// TwinCAT 3 PLC project PLC
// ProgramVersion: 3.1.4023.0
// libraries:
//   Lynus Communicator V2, * (Lynus AG)
//   Lynus Energy Basic, * (Lynus AG)
//   Lynus Energy ModbusTCP, * (Lynus AG)
//   Lynus Persistent Data V1, * (Lynus AG)
//   Tc2_Standard, * (Beckhoff Automation GmbH)
//   Tc2_System, * (Beckhoff Automation GmbH)
//   Tc3_Module, * (Beckhoff Automation GmbH)
// project tree:
//   / Fast.TcTTO, PlcTask.TcTTO, Slow.TcTTO
//   POUs/ prgCom.TcPOU, prgCS1.TcPOU, prgEMS.TcPOU, prgGrid.TcPOU, prgPD.TcPOU, prgVar.TcPOU
// real-time tasks:
//   TASK PlcTask: cycle T#10ms, priority 8, ADS port 350
//   TASK Fast: cycle T#5ms, priority 6, ADS port 351
//   TASK Slow: cycle T#20ms, priority 10, ADS port 352

CONFIGURATION PLC
    RESOURCE PLC ON TwinCAT3
        TASK Fast(INTERVAL := T#5ms, PRIORITY := 6);
        TASK PlcTask(INTERVAL := T#10ms, PRIORITY := 8);
        TASK Slow(INTERVAL := T#20ms, PRIORITY := 10);
        PROGRAM prgVar WITH Fast : prgVar;
        PROGRAM prgPD WITH PlcTask : prgPD;
        PROGRAM prgGrid WITH PlcTask : prgGrid;
        PROGRAM prgEMS WITH PlcTask : prgEMS;
        PROGRAM prgCS1 WITH PlcTask : prgCS1;
        PROGRAM prgCom WITH Slow : prgCom;
    END_RESOURCE
END_CONFIGURATION

// ---- POUs/prgVar.TcPOU
PROGRAM prgVar
VAR
	fbVar			: FB_VarInfo;
	fbrw1			: FB_ReadWrite;
END_VAR

fbVar(
	bReadInfo:= , 
	eTMCFile:= eSelectTMCFile.eDontUseTMCFile, 
	eSavePositionTMCFile:= eSavePositionOnPLC.ePostionHardDisk, 
	udiCounterFoundVariables=> , 
	bError=> , 
	bBusy=> , 
	byProgress=> , 
	udiErrorCodeOut=> , 
	eErrorVarInfo_Out=> , 
	sVarWithError=> );
	
fbrw1();

END_PROGRAM

// ---- POUs/prgPD.TcPOU
PROGRAM prgPD
VAR
	fbPers						: FB_WritePersistentData_CX81xx;
END_VAR

fbPers(
	eSaveModeData:= eUSVSaveMode.eSaveWhenPowerfail, 
	bLoadPersistentDataOk=> , 
	bPowerFailDetect=> , 
	bError=> , 
	bySaveProcess=> , 
	dwStorageLast24h=> , 
	udiErrorCode=> );

END_PROGRAM

// ---- POUs/prgGrid.TcPOU
PROGRAM prgGrid
VAR PERSISTENT
	rSizeGridConn				: REAL;									//{#lynus.ag#()}
END_VAR
VAR
	fbGrid						: FB_Grid_Power_Ext_Input;
	lrGridPower					: LREAL;								//{#lynus.ag#()}
END_VAR

IF prgCS1.byErrorWarningDC_1 = 2 THEN fbGrid.bExtErrorGrid := TRUE; ELSE fbGrid.bExtErrorGrid := FALSE; END_IF

fbGrid(
	bEnable:= TRUE, 
	diNrOfEMS_IN:= prgEMS.fbEMS.diNrOfEMS_OUT, 
	rSizeGridConn:= rSizeGridConn, 
	bExtErrorGrid:= , 
	lrExtGridPower:= prgCS1.fbApliT_1.lrTotalPowerECSRealTime, 
	lrExtTotalCounterEnergy_Consumption:= 0, 
	lrExtTotalCounterEnergy_Production:= 0, 
	lrExtCounterEnergyT1_Consumption:= 0, 
	lrExtCounterEnergyT2_Consumption:= 0, 
	lrExtCounterEnergyT1_Production:= 0, 
	lrExtCounterEnergyT2_Production:= 0, 
	stDataGrid=> , 
	diNrOfGrid_OUT=> );
	
lrGridPower := fbGrid.stDataGrid.lrPower;

END_PROGRAM

// ---- POUs/prgCS1.TcPOU
PROGRAM prgCS1
VAR
	fbApliT_1					: FB_ECS_Alpitronic_Hypercharger;
	
	bSManualyOn_DC_1			: BOOL;												//{#lynus.ag#()}
	bEnabled					: BOOL;												//{#lynus.ag#()}
	bySManualyTargetPowerDC_1	: BYTE;												//{#lynus.ag#()}
	bySMinPowerECSDC_1			: BYTE;												//{#lynus.ag#()}
	byErrorWarningDC_1			: BYTE;												//{#lynus.ag#()}
	lrPowerTotalDC1				: LREAL;											//{#lynus.ag#()}
	lrPowerDC1_S1				: LREAL;											//{#lynus.ag#()}
	lrPowerDC1_S2				: LREAL;											//{#lynus.ag#()}
	lrPowerDC1_S3				: LREAL;											//{#lynus.ag#()}
	rChargingTimeInMinDC1_S1	: REAL;												//{#lynus.ag#()}
	rChargingTimeInMinDC1_S2	: REAL;												//{#lynus.ag#()}
	rChargingTimeInMinDC1_S3	: REAL;												//{#lynus.ag#()}
	rTargetPowerDC1				: REAL;												//{#lynus.ag#()}
	dwSOCCarDC1_S1				: DWORD;											//{#lynus.ag#()}
	dwSOCCarDC1_S2				: DWORD;											//{#lynus.ag#()}
	wStateDC1_S1				: WORD;												//{#lynus.ag#()}
	wStateDC1_S2				: WORD;												//{#lynus.ag#()}
	wStateDC1_S3				: WORD;												//{#lynus.ag#()}
	lrEnergySessionDC1_S1		: LREAL;											//{#lynus.ag#()}
	lrEnergySessionDC1_S2		: LREAL;											//{#lynus.ag#()}
	lrEnergySessionDC1_S3		: LREAL;											//{#lynus.ag#()}
	lrTotalEnergyDC1			: LREAL;											//{#lynus.ag#()}
END_VAR
VAR PERSISTENT
	bEnableDC1					: BOOL;												//{#lynus.ag#()}
	bManualyOnDC_1				: BOOL;												//{#lynus.ag#()}
	byMinPowerDC1				: BYTE;												//{#lynus.ag#()}
	byManualyTargetPowerDC_1	: BYTE;												//{#lynus.ag#()}
	byPrioDC1					: BYTE;												//{#lynus.ag#()}
	bySOCEnableDC1				: BYTE;												//{#lynus.ag#()}
	bySOCDisableDC1				: BYTE;												//{#lynus.ag#()}
	rMaxPowerDC1				: REAL;												//{#lynus.ag#()}
END_VAR

//Manual Power
fbApliT_1.stSetupECS.bManualyOn := bManualyOnDC_1;
	fbApliT_1.stSetupECS.byManualyTargetPower := byManualyTargetPowerDC_1;
		fbApliT_1.stSetupECS.byPriority := byPrioDC1;
			fbApliT_1.stSetupECS.byEnableSOC := bySOCEnableDC1;
				fbApliT_1.stSetupECS.byDisableSOC := bySOCDisableDC1;
					fbApliT_1.stSetupECS.rMaxPower := rMaxPowerDC1;
						fbApliT_1.stSetupECS.byCSMinPower := byMinPowerDC1;	
	
fbApliT_1(
	bEnable:= bEnableDC1, 
	bPowerDataInvers:= , 
	byElectricFuseLine:= , 
	byUnitID:= 1, 
	diNrOfEMS_IN:= prgEMS.fbEMS.diNrOfEMS_OUT, 
	diNrOfEM_IN_CS:= , 
	sIPAdress:= '192.168.1.100', 
	stSetupECS:= , 
	stDataECS=> , 
	diNrOfECS_OUT=> );

bSManualyOn_DC_1 := fbApliT_1.stDataECS.bSManualyOn;
	bySManualyTargetPowerDC_1 := fbApliT_1.stDataECS.bySManualyTargetPower;
		byErrorWarningDC_1 := fbApliT_1.stDataECS.byErrorWarning;
			lrPowerTotalDC1 := fbApliT_1.stDataECS.lrTotalPower;
				lrPowerDC1_S1 :=  fbApliT_1.stDataECS.arrSocketPower[1];
					lrPowerDC1_S2 :=  fbApliT_1.stDataECS.arrSocketPower[2];
						lrPowerDC1_S3 := fbApliT_1.stDataECS.arrSocketPower[3];	 	
							rChargingTimeInMinDC1_S1 := fbApliT_1.stDataECS.arrChargingTimeInMin[1];	
								rChargingTimeInMinDC1_S2 := fbApliT_1.stDataECS.arrChargingTimeInMin[2];
									rChargingTimeInMinDC1_S3 := fbApliT_1.stDataECS.arrChargingTimeInMin[3];
										dwSOCCarDC1_S1 := fbApliT_1.stDataECS.arrSocketSOCCar[1]; 
											dwSOCCarDC1_S2 := fbApliT_1.stDataECS.arrSocketSOCCar[2]; 	
												wStateDC1_S1 := fbApliT_1.stDataECS.arrSocketStateECS[1];
													wStateDC1_S2 := fbApliT_1.stDataECS.arrSocketStateECS[2];
														wStateDC1_S3 := fbApliT_1.stDataECS.arrSocketStateECS[3];
															lrEnergySessionDC1_S1 := fbApliT_1.stDataECS.arrSocketEnergySession[1];
																lrEnergySessionDC1_S2 := fbApliT_1.stDataECS.arrSocketEnergySession[2];
																	lrEnergySessionDC1_S3 := fbApliT_1.stDataECS.arrSocketEnergySession[3];
																		lrTotalEnergyDC1 := fbApliT_1.stDataECS.lrTotalCounterEnergy_Consumption;
																			bySMinPowerECSDC_1 := fbApliT_1.stDataECS.bySCSMinPower;
																				rTargetPowerDC1 := fbApliT_1.stDataECS.rTargetPower;
																					bEnabled := fbApliT_1.stDataECS.bEnabled;

END_PROGRAM

// ---- POUs/prgEMS.TcPOU
PROGRAM prgEMS
VAR PERSISTENT
	byMaxDepthOfDischrgEPO		: BYTE;							//{#lynus.ag#()}
	byPrioMinChrgBattSOCInEPO	: BYTE;							//{#lynus.ag#()}
	byResChrgfromGridToBatt		: BYTE;							//{#lynus.ag#()}
	byReserveSOCEPO				: BYTE;							//{#lynus.ag#()}
	uiUpdateTime				: UINT;							//{#lynus.ag#()}
	bEnableEMS					: BOOL;							//{#lynus.ag#()}
	bEnableMainFuse				: BOOL;							//{#lynus.ag#()}
	bAllowChrgFromGrid			: BOOL;							//{#lynus.ag#()}
	rMainFuseCSEMS				: REAL;							//{#lynus.ag#()}
	iOperationModeEMS			: INT;							//{#lynus.ag#()}
END_VAR
VAR
	fbEMS						: FB_EMS_V2;
	bIsEnableEMS				: BOOL;							//{#lynus.ag#()}
	bStateAllowChrgFromGrid		: BOOL;							//{#lynus.ag#()}
	bHPActivate					: BOOL;							//{#lynus.ag#()}
	bControllingState			: BOOL;							//{#lynus.ag#()}
	bSEnableMainFuse			: BOOL;							//{#lynus.ag#()}
	iMessageEMS					: INT;							//{#lynus.ag#()}
	rHeartbeatEMS				: REAL;							//{#lynus.ag#()}
	rErrorWarningEMS			: REAL;							//{#lynus.ag#()}
	rReadyEMS					: REAL;							//{#lynus.ag#()}
	rNewBatteryPowerEMS			: REAL;							//{#lynus.ag#()}
END_VAR

fbEMS.stSetupEMS.bAllowChrgFromGrid := bAllowChrgFromGrid;
	fbEMS.stSetupEMS.byMaxDepthOfDischrgEPO := byMaxDepthOfDischrgEPO;
		fbEMS.stSetupEMS.byPrioChrgBattSOCInEPO := byPrioMinChrgBattSOCInEPO;
			fbEMS.stSetupEMS.byResChrgGridToBatt := byResChrgfromGridToBatt;
				fbEMS.stSetupEMS.byReserveSOCEPO := byReserveSOCEPO;
					fbEMS.stSizeMainFuseCS.rElSizeLine1 := rMainFuseCSEMS;
						fbEMS.stSetupEMS.uiUpdateTime := uiUpdateTime;
							fbEMS.stSetupEMS.bEnableMainFuseFunc := bEnableMainFuse;

IF iOperationModeEMS = 0 THEN fbEMS.eOperationMode := E_OperatingMode_EMS.eAllOff;
ELSIF iOperationModeEMS = 1 THEN fbEMS.eOperationMode := E_OperatingMode_EMS.eSelfConsumption;	
ELSIF iOperationModeEMS = 2 THEN fbEMS.eOperationMode := E_OperatingMode_EMS.ePeakLoadCapping;
ELSIF iOperationModeEMS = 3 THEN fbEMS.eOperationMode := E_OperatingMode_EMS.eLoadManagement;			
END_IF

fbEMS(
	bEnable:= bEnableEMS, 
	tDelayPwrCorrectionECS:= T#2.5S, 
	stNrOfEM_IN_ECS:= , 
	stSizeMainFuseCS:= , 
	stSetupEMS:= , 
	eOperationMode:= , 
	eSpeedModeBackendController:= E_SpeedModeBackendController_EMS.eSlow, 
	eSpeedModeLocalController:= E_SpeedModeLocalController_EMS.eSlow,
	bActivateHP:= bHPActivate, 
	bControllingState:= bControllingState, 
	rHeartbeat:= rHeartbeatEMS, 
	rErrorWarning:= rErrorWarningEMS, 
	rEnergyOptReady:= rReadyEMS, 
	rNewBattPower:= rNewBatteryPowerEMS, 
	eMessageEMS=> iMessageEMS, 
	bStateEnable=> bIsEnableEMS, 
	bStateAllowChrgFromGrid=> bStateAllowChrgFromGrid, 
	bMissingPowerData=> , 
	bSurplusAvailable=> , 
	bSEnableMainFuseFunc=> bSEnableMainFuse, 
	byProgress=> , 
	uiState_OUT=> , 
	diNrOfEMS_OUT=> , 
	arrMinPrioReached=> , 
	arrMaxPrioReached=> );

END_PROGRAM

// ---- POUs/prgCom.TcPOU
PROGRAM prgCom
VAR
	fbCom			: FB_MqttCommunicator;
END_VAR

fbCom(
	bConnect:= TRUE, 
	sUserName:= 'a72d1e6c-755b-4f3d-bd19-1d4ef4a76d7b', 
	sUserPassword:= '18d6ab8a-4f65-4c49-9d83-db4a7e229b05', 
	eSavePositionCertificate:= eSavePositionOnPLC.ePostionHardDisk, 
	bConnected=> , 
	bError=> , 
	hrErrorCode=> , 
	eConnectionState=> , 
	eErrorMessage_Out=> );

END_PROGRAM
